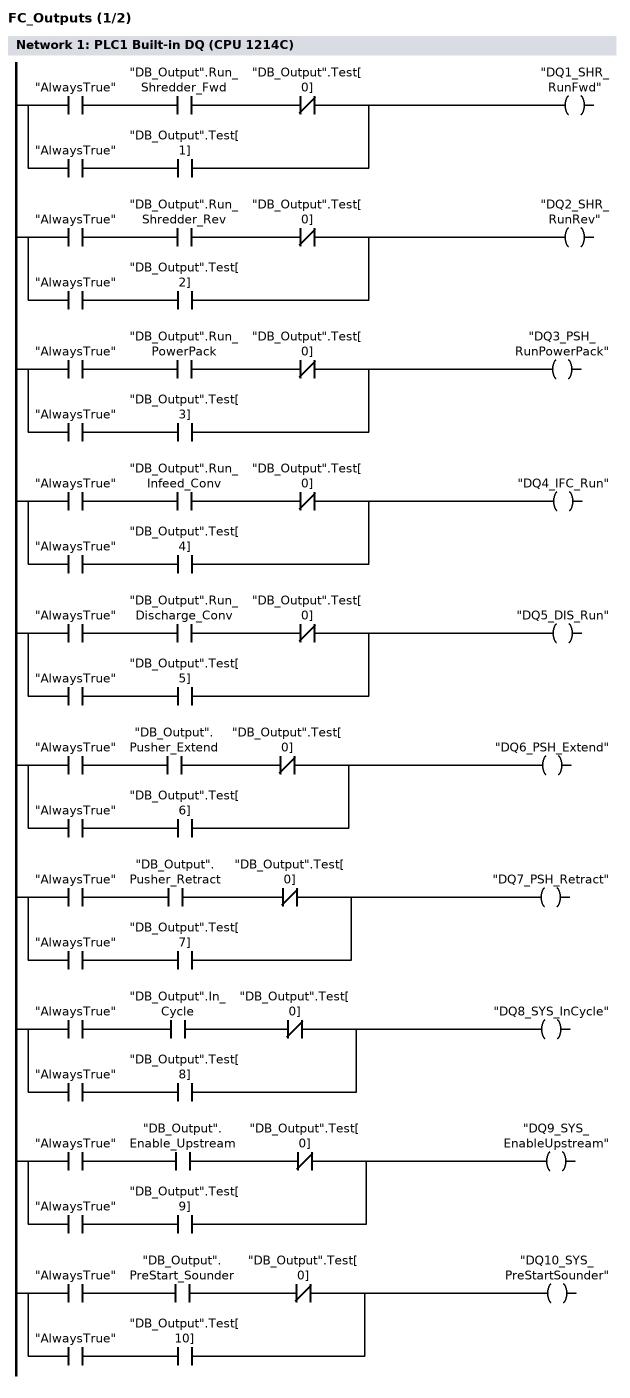
   RUNG wire#powerrail
      Contact( "AlwaysTrue" )
      Contact( "DB_Output".Run_Shredder_Fwd )
      I_Contact( "DB_Output".Test[0] )
      wire#w1
      Coil( "DQ1_SHR_RunFwd" )
   END_RUNG
   RUNG wire#powerrail
      Contact( "AlwaysTrue" )
      Contact( "DB_Output".Test[1] )
   END_RUNG wire#w1
   RUNG wire#powerrail
      Contact( "AlwaysTrue" )
      Contact( "DB_Output".Run_Shredder_Rev )
      I_Contact( "DB_Output".Test[0] )
      wire#w2
      Coil( "DQ2_SHR_RunRev" )
   END_RUNG
   RUNG wire#powerrail
      Contact( "AlwaysTrue" )
      Contact( "DB_Output".Test[2] )
   END_RUNG wire#w2
   RUNG wire#powerrail
      Contact( "AlwaysTrue" )
      Contact( "DB_Output".Run_PowerPack )
      I_Contact( "DB_Output".Test[0] )
      wire#w3
      Coil( "DQ3_PSH_RunPowerPack" )
   END_RUNG
   RUNG wire#powerrail
      Contact( "AlwaysTrue" )
      Contact( "DB_Output".Test[3] )
   END_RUNG wire#w3
   RUNG wire#powerrail
      Contact( "AlwaysTrue" )
      Contact( "DB_Output".Run_Infeed_Conv )
      I_Contact( "DB_Output".Test[0] )
      wire#w4
      Coil( "DQ4_IFC_Run" )
   END_RUNG
   RUNG wire#powerrail
      Contact( "AlwaysTrue" )
      Contact( "DB_Output".Test[4] )
   END_RUNG wire#w4
   RUNG wire#powerrail
      Contact( "AlwaysTrue" )
      Contact( "DB_Output".Run_Discharge_Conv )
      I_Contact( "DB_Output".Test[0] )
      wire#w5
      Coil( "DQ5_DIS_Run" )
   END_RUNG
   RUNG wire#powerrail
      Contact( "AlwaysTrue" )
      Contact( "DB_Output".Test[5] )
   END_RUNG wire#w5
   RUNG wire#powerrail
      Contact( "AlwaysTrue" )
      Contact( "DB_Output".Pusher_Extend )
      I_Contact( "DB_Output".Test[0] )
      wire#w6
      Coil( "DQ6_PSH_Extend" )
   END_RUNG
   RUNG wire#powerrail
      Contact( "AlwaysTrue" )
      Contact( "DB_Output".Test[6] )
   END_RUNG wire#w6
   RUNG wire#powerrail
      Contact( "AlwaysTrue" )
      Contact( "DB_Output".Pusher_Retract )
      I_Contact( "DB_Output".Test[0] )
      wire#w7
      Coil( "DQ7_PSH_Retract" )
   END_RUNG
   RUNG wire#powerrail
      Contact( "AlwaysTrue" )
      Contact( "DB_Output".Test[7] )
   END_RUNG wire#w7
   RUNG wire#powerrail
      Contact( "AlwaysTrue" )
      Contact( "DB_Output".In_Cycle )
      I_Contact( "DB_Output".Test[0] )
      wire#w8
      Coil( "DQ8_SYS_InCycle" )
   END_RUNG
   RUNG wire#powerrail
      Contact( "AlwaysTrue" )
      Contact( "DB_Output".Test[8] )
   END_RUNG wire#w8
   RUNG wire#powerrail
      Contact( "AlwaysTrue" )
      Contact( "DB_Output".Enable_Upstream )
      I_Contact( "DB_Output".Test[0] )
      wire#w9
      Coil( "DQ9_SYS_EnableUpstream" )
   END_RUNG
   RUNG wire#powerrail
      Contact( "AlwaysTrue" )
      Contact( "DB_Output".Test[9] )
   END_RUNG wire#w9
   RUNG wire#powerrail
      Contact( "AlwaysTrue" )
      Contact( "DB_Output".PreStart_Sounder )
      I_Contact( "DB_Output".Test[0] )
      wire#w10
      Coil( "DQ10_SYS_PreStartSounder" )
   END_RUNG
   RUNG wire#powerrail
      Contact( "AlwaysTrue" )
      Contact( "DB_Output".Test[10] )
   END_RUNG wire#w10
   // the same network as SCL:
   "DQ1_SHR_RunFwd" := ("AlwaysTrue" AND "DB_Output".Run_Shredder_Fwd AND NOT "DB_Output".Test[0]) OR ("AlwaysTrue" AND "DB_Output".Test[1]);
   "DQ2_SHR_RunRev" := ("AlwaysTrue" AND "DB_Output".Run_Shredder_Rev AND NOT "DB_Output".Test[0]) OR ("AlwaysTrue" AND "DB_Output".Test[2]);
   "DQ3_PSH_RunPowerPack" := ("AlwaysTrue" AND "DB_Output".Run_PowerPack AND NOT "DB_Output".Test[0]) OR ("AlwaysTrue" AND "DB_Output".Test[3]);
   "DQ4_IFC_Run" := ("AlwaysTrue" AND "DB_Output".Run_Infeed_Conv AND NOT "DB_Output".Test[0]) OR ("AlwaysTrue" AND "DB_Output".Test[4]);
   "DQ5_DIS_Run" := ("AlwaysTrue" AND "DB_Output".Run_Discharge_Conv AND NOT "DB_Output".Test[0]) OR ("AlwaysTrue" AND "DB_Output".Test[5]);
   "DQ6_PSH_Extend" := ("AlwaysTrue" AND "DB_Output".Pusher_Extend AND NOT "DB_Output".Test[0]) OR ("AlwaysTrue" AND "DB_Output".Test[6]);
   "DQ7_PSH_Retract" := ("AlwaysTrue" AND "DB_Output".Pusher_Retract AND NOT "DB_Output".Test[0]) OR ("AlwaysTrue" AND "DB_Output".Test[7]);
   "DQ8_SYS_InCycle" := ("AlwaysTrue" AND "DB_Output".In_Cycle AND NOT "DB_Output".Test[0]) OR ("AlwaysTrue" AND "DB_Output".Test[8]);
   "DQ9_SYS_EnableUpstream" := ("AlwaysTrue" AND "DB_Output".Enable_Upstream AND NOT "DB_Output".Test[0]) OR ("AlwaysTrue" AND "DB_Output".Test[9]);
   "DQ10_SYS_PreStartSounder" := ("AlwaysTrue" AND "DB_Output".PreStart_Sounder AND NOT "DB_Output".Test[0]) OR ("AlwaysTrue" AND "DB_Output".Test[10]);
END_REGION

REGION Network 2: PLC1.1 SM1223 DQ Relay
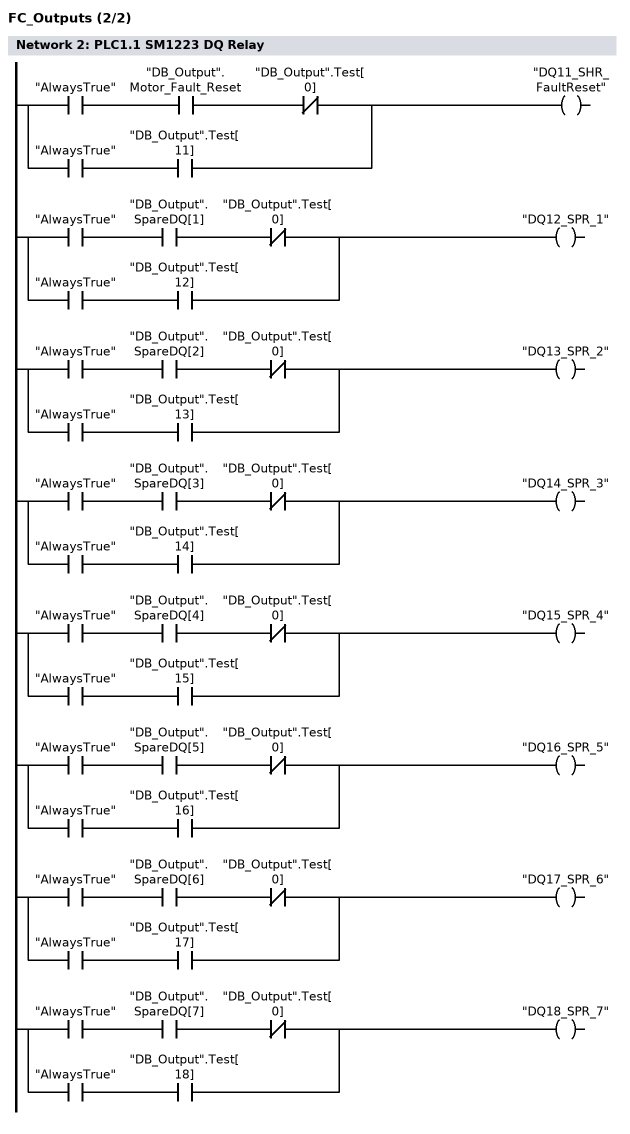
   RUNG wire#powerrail
      Contact( "AlwaysTrue" )
      Contact( "DB_Output".Motor_Fault_Reset )
      I_Contact( "DB_Output".Test[0] )
      wire#w1
      Coil( "DQ11_SHR_FaultReset" )
   END_RUNG
   RUNG wire#powerrail
      Contact( "AlwaysTrue" )
      Contact( "DB_Output".Test[11] )
   END_RUNG wire#w1
   RUNG wire#powerrail
      Contact( "AlwaysTrue" )
      Contact( "DB_Output".SpareDQ[1] )
      I_Contact( "DB_Output".Test[0] )
      wire#w2
      Coil( "DQ12_SPR_1" )
   END_RUNG
   RUNG wire#powerrail
      Contact( "AlwaysTrue" )
      Contact( "DB_Output".Test[12] )
   END_RUNG wire#w2
   RUNG wire#powerrail
      Contact( "AlwaysTrue" )
      Contact( "DB_Output".SpareDQ[2] )
      I_Contact( "DB_Output".Test[0] )
      wire#w3
      Coil( "DQ13_SPR_2" )
   END_RUNG
   RUNG wire#powerrail
      Contact( "AlwaysTrue" )
      Contact( "DB_Output".Test[13] )
   END_RUNG wire#w3
   RUNG wire#powerrail
      Contact( "AlwaysTrue" )
      Contact( "DB_Output".SpareDQ[3] )
      I_Contact( "DB_Output".Test[0] )
      wire#w4
      Coil( "DQ14_SPR_3" )
   END_RUNG
   RUNG wire#powerrail
      Contact( "AlwaysTrue" )
      Contact( "DB_Output".Test[14] )
   END_RUNG wire#w4
   RUNG wire#powerrail
      Contact( "AlwaysTrue" )
      Contact( "DB_Output".SpareDQ[4] )
      I_Contact( "DB_Output".Test[0] )
      wire#w5
      Coil( "DQ15_SPR_4" )
   END_RUNG
   RUNG wire#powerrail
      Contact( "AlwaysTrue" )
      Contact( "DB_Output".Test[15] )
   END_RUNG wire#w5
   RUNG wire#powerrail
      Contact( "AlwaysTrue" )
      Contact( "DB_Output".SpareDQ[5] )
      I_Contact( "DB_Output".Test[0] )
      wire#w6
      Coil( "DQ16_SPR_5" )
   END_RUNG
   RUNG wire#powerrail
      Contact( "AlwaysTrue" )
      Contact( "DB_Output".Test[16] )
   END_RUNG wire#w6
   RUNG wire#powerrail
      Contact( "AlwaysTrue" )
      Contact( "DB_Output".SpareDQ[6] )
      I_Contact( "DB_Output".Test[0] )
      wire#w7
      Coil( "DQ17_SPR_6" )
   END_RUNG
   RUNG wire#powerrail
      Contact( "AlwaysTrue" )
      Contact( "DB_Output".Test[17] )
   END_RUNG wire#w7
   RUNG wire#powerrail
      Contact( "AlwaysTrue" )
      Contact( "DB_Output".SpareDQ[7] )
      I_Contact( "DB_Output".Test[0] )
      wire#w8
      Coil( "DQ18_SPR_7" )
   END_RUNG
   RUNG wire#powerrail
      Contact( "AlwaysTrue" )
      Contact( "DB_Output".Test[18] )
   END_RUNG wire#w8
   // the same network as SCL:
   "DQ11_SHR_FaultReset" := ("AlwaysTrue" AND "DB_Output".Motor_Fault_Reset AND NOT "DB_Output".Test[0]) OR ("AlwaysTrue" AND "DB_Output".Test[11]);
   "DQ12_SPR_1" := ("AlwaysTrue" AND "DB_Output".SpareDQ[1] AND NOT "DB_Output".Test[0]) OR ("AlwaysTrue" AND "DB_Output".Test[12]);
   "DQ13_SPR_2" := ("AlwaysTrue" AND "DB_Output".SpareDQ[2] AND NOT "DB_Output".Test[0]) OR ("AlwaysTrue" AND "DB_Output".Test[13]);
   "DQ14_SPR_3" := ("AlwaysTrue" AND "DB_Output".SpareDQ[3] AND NOT "DB_Output".Test[0]) OR ("AlwaysTrue" AND "DB_Output".Test[14]);
   "DQ15_SPR_4" := ("AlwaysTrue" AND "DB_Output".SpareDQ[4] AND NOT "DB_Output".Test[0]) OR ("AlwaysTrue" AND "DB_Output".Test[15]);
   "DQ16_SPR_5" := ("AlwaysTrue" AND "DB_Output".SpareDQ[5] AND NOT "DB_Output".Test[0]) OR ("AlwaysTrue" AND "DB_Output".Test[16]);
   "DQ17_SPR_6" := ("AlwaysTrue" AND "DB_Output".SpareDQ[6] AND NOT "DB_Output".Test[0]) OR ("AlwaysTrue" AND "DB_Output".Test[17]);
   "DQ18_SPR_7" := ("AlwaysTrue" AND "DB_Output".SpareDQ[7] AND NOT "DB_Output".Test[0]) OR ("AlwaysTrue" AND "DB_Output".Test[18]);
END_REGION
END_FUNCTION

DATA_BLOCK "iDB_MotorFwdRevSystem_Shredder"   // DB6
VERSION : 0.1
// stored: AutoNumber true, DBAccessibleFromOPCUA true, InstanceOfName FB_MotorFwdRevSystem, InstanceOfType FB
"FB_MotorFwdRevSystem"
BEGIN
   IO.ReverseDelay := 8.0;
END_DATA_BLOCK

DATA_BLOCK "iDB_PusherControl"   // DB10
VERSION : 0.1
// stored: AutoNumber true, DBAccessibleFromOPCUA true, InstanceOfName FB_PusherControl, InstanceOfType FB
"FB_PusherControl"
BEGIN
END_DATA_BLOCK

DATA_BLOCK "iDB_ShredderSequencer"   // DB11
VERSION : 0.1
// stored: AutoNumber true, DBAccessibleFromOPCUA true, InstanceOfName FB_ShredderSequencer, InstanceOfType FB
"FB_ShredderSequencer"
BEGIN
END_DATA_BLOCK
